PROGRAM MAIN
VAR
END_VAR

PRG_EM1K0_GMD_VGC_1();
PRG_GMD();
PRG_TV1K0_GAS_VGC_1();

END_PROGRAM

(* stored: Version 1.1.0.1, ProductVersion 3.1.4022.12
   POU MAIN: Id {80634dbc-d649-47af-a183-d3f1342ca1c9}, SpecialFunc None *)
